// TIA Portal V20 export
// export: Created 2025-12-01T14:56:13.8711928Z, ExportSetting None, DisplayName Totally Integrated Automation Portal, DisplayVersion V20 Update 3, DisplayName TIA Portal Openness, DisplayVersion V20 Update 3, DisplayName TIA Portal Version Control Interface, DisplayVersion V20 Update 3, DisplayName STEP 7 Professional, DisplayVersion V20 Update 3, DisplayName STEP 7 Safety, DisplayVersion V20 Update 2, DisplayName WinCC Basic/Comfort/Advanced, DisplayVersion V20 Update 3, DisplayName WinCC Professional, DisplayVersion V20 Update 3, DisplayName WinCC Unified, DisplayVersion V20 Update 3
TYPE "UDT_UTs_Control"
   STRUCT
      UT_AnteriorMesa : UInt;   // UT Anterior dentro de la Mesa
      UT_SiguienteMesa : UInt;   // UT Siguiente dentro de la Mesa
      EstadoRecepcionUT : UInt;   // Estado de Tratamiento de la Recepción de la UT
      EstadoEmisionUT : UInt;   // Estado de Tratamiento de la Emisión de la UT
      EstadoGeneralUT : UInt;   // Estado de Tratamiento de Petición de Eventos a Generar
      EstadoEventoRecibido : UInt;   // Estado de Eventos Recibidos
      EstadoEventoAGenerar : UInt;   // Estado de Eventos A Generar
      Mckey : UDInt;   // McKey de la UT
      MesaActual : UInt;   // Mesa Actual de la UT
      MesaDestino : UInt;   // Mesa Destino de la UT
      MesaIntermedia : UInt;   // Mesa Intermedia de la UT
      Grupo : UInt;   // Numero de Grupo de la UT
      CantidadGrupo : USInt;   // Cantidad de UT's del Grupo
      PosicionGrupo : USInt;   // Posicion de la UT en el Grupo
      TipoCarga : USInt;   // Tipo de Carga (Euro,Caja, Remo ...)
      AtributosDelaCarga : Struct
         Vacia : Bool;   // Atributos Especiales del la Carga --> Vacia
         Pila : Bool;   // Atributos Especiales del la Carga --> Pila
         Remontada : Bool;   // Atributos Especiales del la Carga --> Remontada
      END_STRUCT;
      AtributosDeLaUT : Struct
         MemorizarRETI : Bool;   // Atributos de la UT --> Memorizar recibido el RETI (Salida MesaIntermedia)
         RecircularCarga : Bool;   // Atributos de la UT --> Recicular la Carga (RUTA)
         PeticionDeDatos : Bool;   // Atributos de la UT --> Pedir Datos (DAT?)
         LadoDeLaEtiqueta : Bool;   // Atributos de la UT --> Lado donde esta la Etiqueta (Derecha / Izquierda)
      END_STRUCT;
      EventosDeCambioDeMesa : Struct
         PeticionCambiarUTDeMesa : Bool;   // Atributos de Cambio de Mesa -> Peticion de Cambio de Mesa
         NOKCambiarUTDeMesa : Bool;   // Atributos de Cambio de Mesa -> No Cambiar de Mesa
         OKCambiarUTDeMesaInicio : Bool;   // Atributos de Cambio de Mesa -> Cambiar de Mesa al Inicio
         OKCambiarUTDeMesaFinal : Bool;   // Atributos de Cambio de Mesa -> Cambiar de Mesa al Final
      END_STRUCT;
      EventosInformarJdT : Struct
         DuplicidadMckey : Bool;   // Atributos de Informe para el JdT -> Duplicidad de Mckey (CREA)
         CambiadaDeMesa : Bool;   // Atributos de Informe para el JdT -> Cambiada de Mesa
         NoCambidaDeMesa : Bool;   // Atributos de Informe para el JdT -> No Cambiada de Mesa
         CambiadaPosicionDown : Bool;   // Atributos de Informe para el JdT -> Cambiada de Posicion Down en Mesa
         CambiadaPosicionUp : Bool;   // Atributos de Informe para el JdT -> Cambiada de Posicion Up en Mesa
         PeticionDeDatos : Bool;
         ChequeoDelReset : Bool;
      END_STRUCT;
   END_STRUCT;
END_TYPE
